// Mitsubishi GX Works2 project: EXC_PLC2   PLC: FX3G

// global labels: Global1
VAR_GLOBAL
  StartBtn AT X001 : BOOL;
  AnalogIn AT D8280 : INT;
  SampledValue AT D2000 : REAL;
  IsRegular AT M50 : BOOL;
  IsPremium AT M51 : BOOL;
  RaspberryStock AT D1100 : REAL;
  LemonStock AT D1110 : REAL;
  StabilizerStock AT D1120 : REAL;
  GummyStock AT D1130 : REAL;
  HasStockRegular AT M80 : BOOL;
  HasStockPremium AT M61 : BOOL;
  HasRaspberryStock AT M222 : BOOL;
  HasLemonStock AT M223 : BOOL;
  HasStabilizerStock AT M224 : BOOL;
  HasGummyStock AT M225 : BOOL;
  HasRasprerryStock1 AT M33 : BOOL;
  HasLemonStock1 AT M34 : BOOL;
  HasStabilizerStock1 AT M35 : BOOL;
  HasGummyStock1 AT M36 : BOOL;
  InvalidOrder AT M66 : BOOL;
  Start_Day AT X007 : BOOL;
  Emergency_Stop AT X005 : BOOL;
  System_On_Lamp AT Y007 : BOOL;
  Analog_Output_Value AT D8282 : INT;
  Produced_Packages_Counter AT D4000 : REAL;  (* מונה מארזים בתחילת כל יום מתאפס לאפס *)
  No_Stock_Error AT M20 : BOOL;
  User_valid AT M12 : BOOL;
  Raspberry_User AT D2100 : REAL;
  Lemon_User AT D2110 : REAL;
  Stabilizer_User AT D2120 : REAL;
  Gummy_User AT D2130 : REAL;
END_VAR
VAR_GLOBAL CONSTANT
  C_R_Raspberry : REAL := 280;
  C_R_Lemon : REAL := 455;
  C_R_Stabilizer : REAL := 105;
  C_P_Raspberry : REAL := 385;
  C_P_Lemon : REAL := 665;
  C_P_Stabilizer : REAL := 210;
  C_R_Gummy : REAL := 28;
  C_P_Gummy : REAL := 70;
END_VAR
VAR_GLOBAL
  PreparationActive AT M101 : BOOL;
  PreparationFinished AT M102 : BOOL;
  CoolingActive AT M103 : BOOL;
  TC50 AT TS50 : BOOL;
  TC80 AT TS80 : BOOL;
  StartMixing AT M2 : BOOL;
  TC2 AT TS2 : BOOL;
  TC1 AT TS1 : BOOL;
END_VAR

// task Task_01 (event TRUE, interval 0, priority 31): POU_01

PROGRAM POU_01
(* structured ladder/FBD written out as ST: instructions are called as NAME(EN, inputs, outputs); _pN, _eN, _tN stand for wires *)
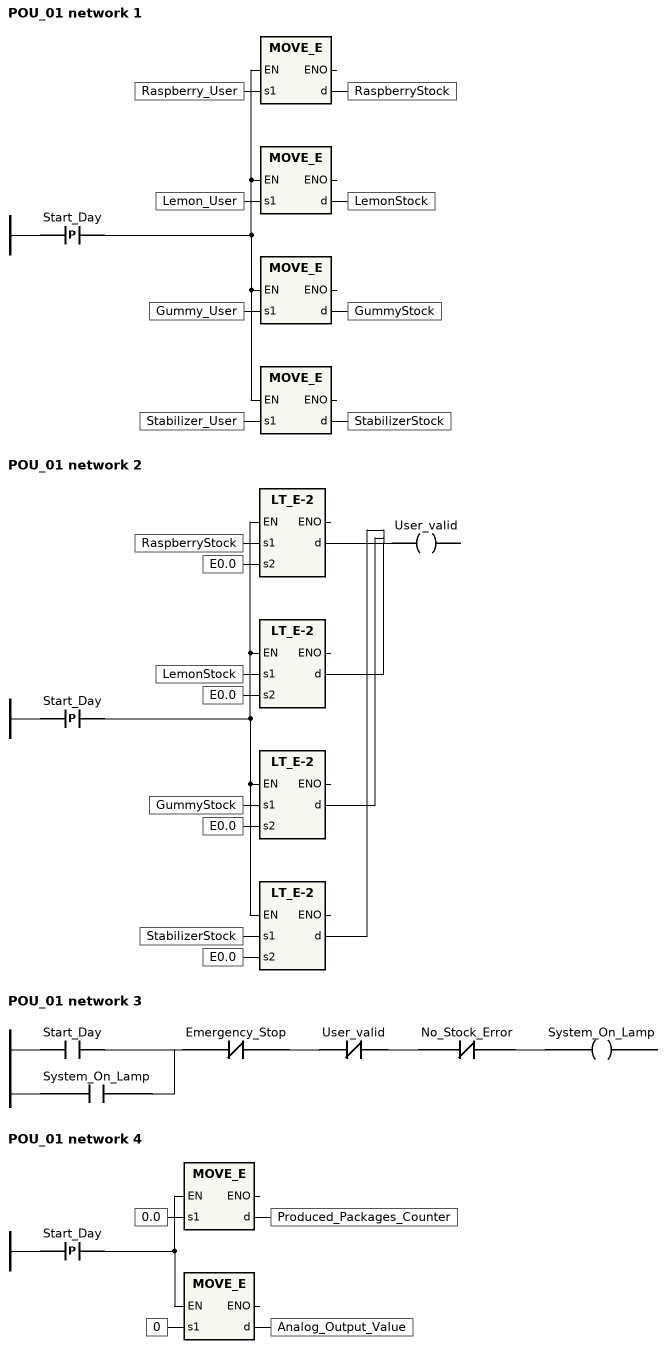
(* network 1 *)
_p1 := LDP(TRUE, Start_Day);
MOVE_E(_p1, Raspberry_User, RaspberryStock);
MOVE_E(_p1, Lemon_User, LemonStock);
MOVE_E(_p1, Gummy_User, GummyStock);
MOVE_E(_p1, Stabilizer_User, StabilizerStock);
(* network 2 *)
_p1 := LDP(TRUE, Start_Day);
LT_E(_p1, RaspberryStock, E0.0, _t2);
LT_E(_p1, LemonStock, E0.0, _t3);
LT_E(_p1, GummyStock, E0.0, _t4);
LT_E(_p1, StabilizerStock, E0.0, _t5);
User_valid := _t2 OR _t3 OR _t4 OR _t5;
(* network 3 *)
System_On_Lamp := (((Start_Day OR System_On_Lamp) AND NOT Emergency_Stop) AND NOT User_valid) AND NOT No_Stock_Error;
(* network 4 *)
_p1 := LDP(TRUE, Start_Day);
MOVE_E(_p1, 0.0, Produced_Packages_Counter);
MOVE_E(_p1, 0, Analog_Output_Value);
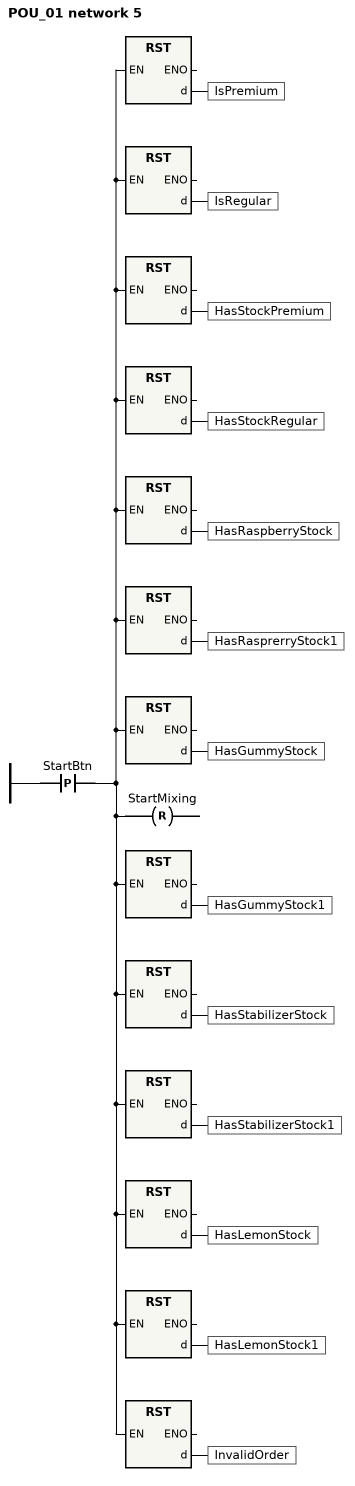
(* network 5 *)
_p1 := LDP(TRUE, StartBtn);
RST(_p1, IsPremium);
RST(_p1, IsRegular);
RST(_p1, HasStockPremium);
RST(_p1, HasStockRegular);
RST(_p1, HasRaspberryStock);
RST(_p1, HasRasprerryStock1);
RST(_p1, HasGummyStock);
RST(_p1, HasGummyStock1);
RST(_p1, HasStabilizerStock);
RST(_p1, HasStabilizerStock1);
RST(_p1, HasLemonStock);
RST(_p1, HasLemonStock1);
RST(_p1, InvalidOrder);
RST(_p1, StartMixing);
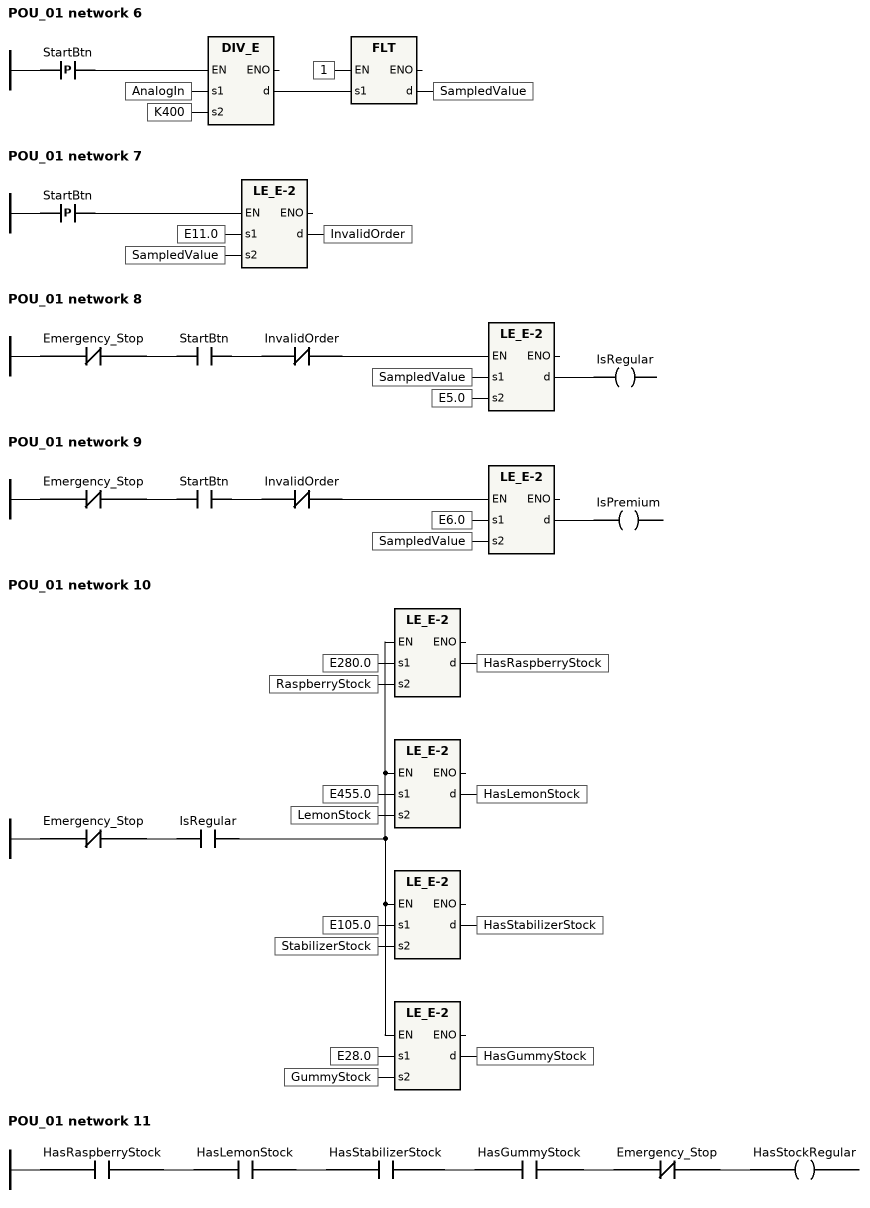
(* network 6 *)
DIV_E(LDP(TRUE, StartBtn), AnalogIn, K400, _t1);
FLT(1, _t1, SampledValue);
(* network 7 *)
LE_E(LDP(TRUE, StartBtn), E11.0, SampledValue, InvalidOrder);
(* network 8 *)
LE_E(NOT Emergency_Stop AND StartBtn AND NOT InvalidOrder, SampledValue, E5.0, _t1);
IsRegular := _t1;
(* network 9 *)
LE_E(NOT Emergency_Stop AND StartBtn AND NOT InvalidOrder, E6.0, SampledValue, _t1);
IsPremium := _t1;
(* network 10 *)
_p1 := NOT Emergency_Stop AND IsRegular;
LE_E(_p1, E280.0, RaspberryStock, HasRaspberryStock);
LE_E(_p1, E455.0, LemonStock, HasLemonStock);
LE_E(_p1, E105.0, StabilizerStock, HasStabilizerStock);
LE_E(_p1, E28.0, GummyStock, HasGummyStock);
(* network 11 *)
HasStockRegular := HasRaspberryStock AND HasLemonStock AND HasStabilizerStock AND HasGummyStock AND NOT Emergency_Stop;
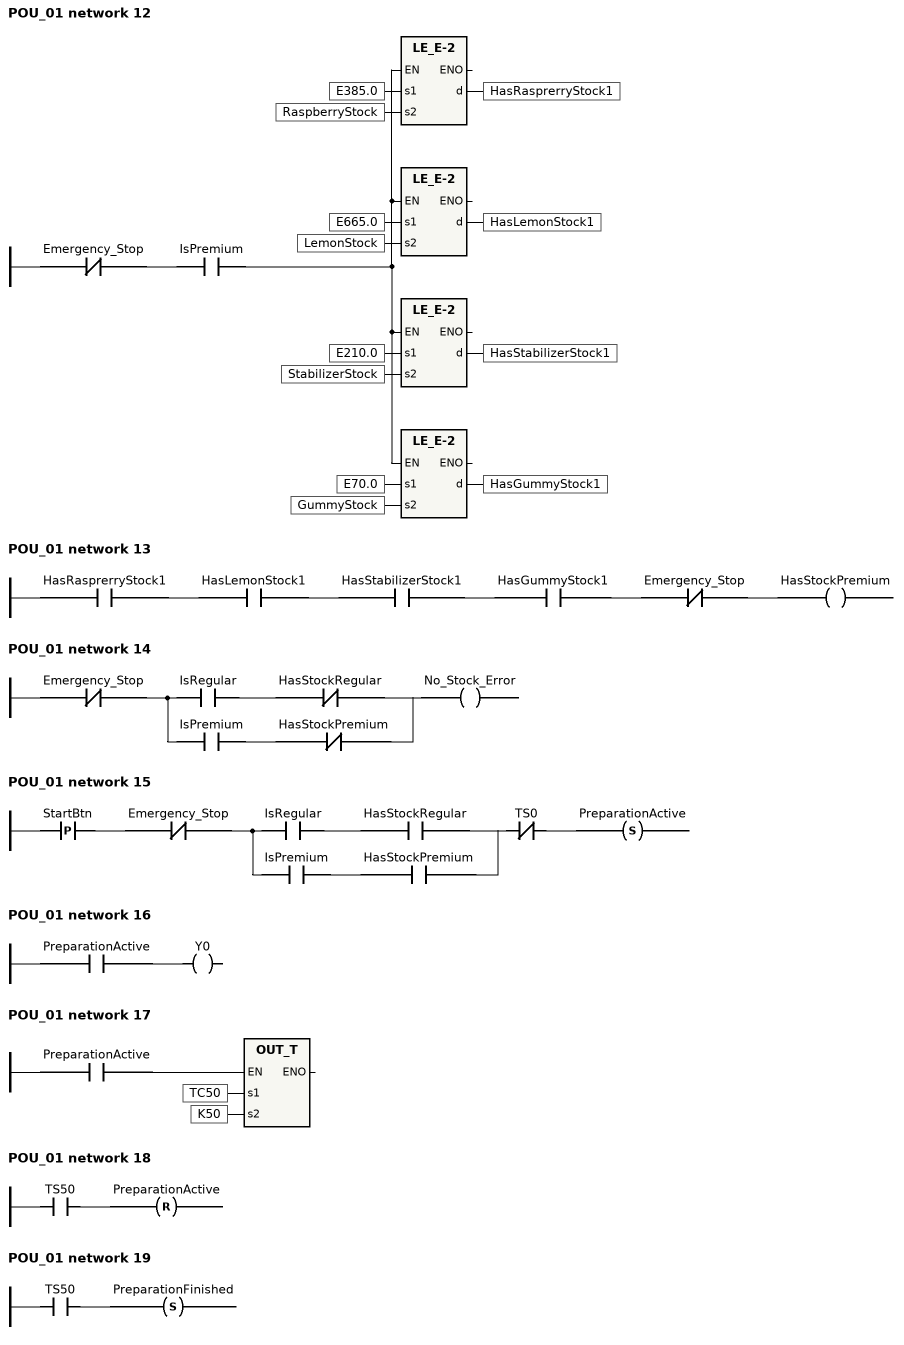
(* network 12 *)
_p1 := NOT Emergency_Stop AND IsPremium;
LE_E(_p1, E385.0, RaspberryStock, HasRasprerryStock1);
LE_E(_p1, E665.0, LemonStock, HasLemonStock1);
LE_E(_p1, E210.0, StabilizerStock, HasStabilizerStock1);
LE_E(_p1, E70.0, GummyStock, HasGummyStock1);
(* network 13 *)
HasStockPremium := HasRasprerryStock1 AND HasLemonStock1 AND HasStabilizerStock1 AND HasGummyStock1 AND NOT Emergency_Stop;
(* network 14 *)
_p1 := NOT Emergency_Stop;
No_Stock_Error := (_p1 AND IsRegular AND NOT HasStockRegular) OR (_p1 AND IsPremium AND NOT HasStockPremium);
(* network 15 *)
_p1 := LDP(TRUE, StartBtn) AND NOT Emergency_Stop;
SET(((_p1 AND IsRegular AND HasStockRegular) OR (_p1 AND IsPremium AND HasStockPremium)) AND NOT TS0, PreparationActive);
(* network 16 *)
Y0 := PreparationActive;
(* network 17 *)
OUT_T(PreparationActive, TC50, K50);
(* network 18 *)
RST(TS50, PreparationActive);
(* network 19 *)
SET(TS50, PreparationFinished);
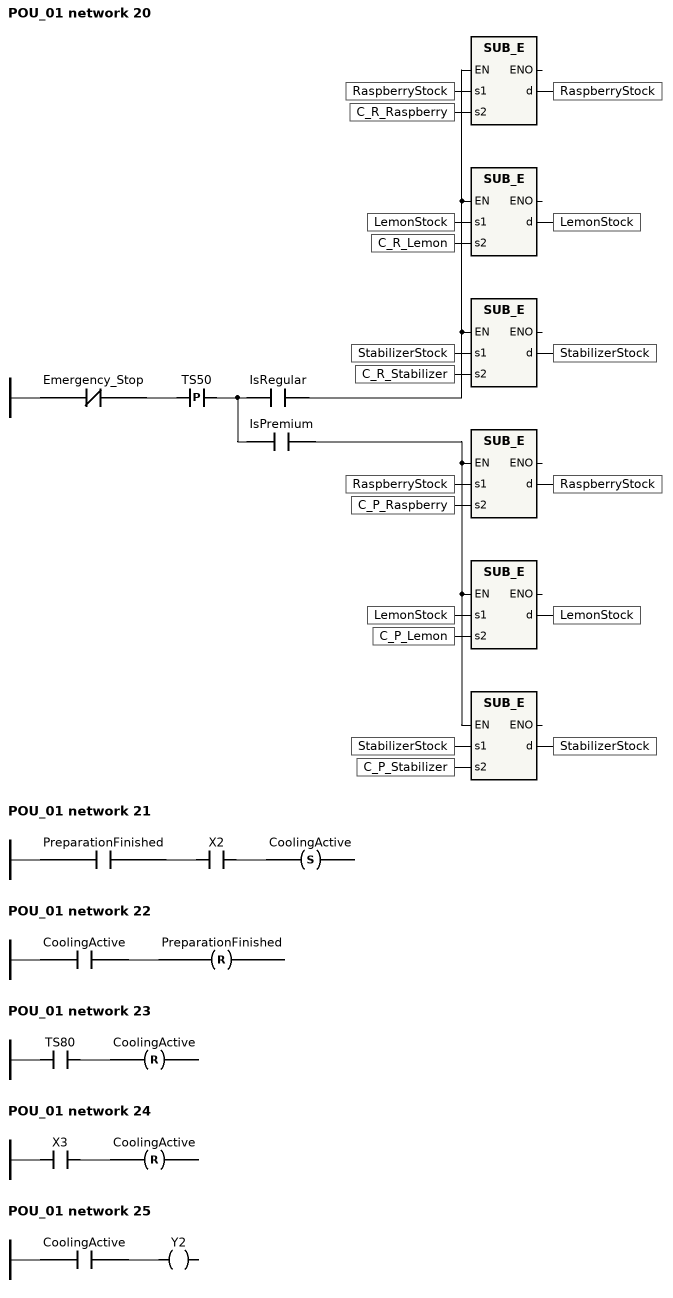
(* network 20 *)
_p1 := NOT Emergency_Stop AND LDP(TRUE, TS50);
_p2 := _p1 AND IsRegular;
SUB_E(_p2, RaspberryStock, C_R_Raspberry, RaspberryStock);
SUB_E(_p2, LemonStock, C_R_Lemon, LemonStock);
SUB_E(_p2, StabilizerStock, C_R_Stabilizer, StabilizerStock);
_p3 := _p1 AND IsPremium;
SUB_E(_p3, RaspberryStock, C_P_Raspberry, RaspberryStock);
SUB_E(_p3, LemonStock, C_P_Lemon, LemonStock);
SUB_E(_p3, StabilizerStock, C_P_Stabilizer, StabilizerStock);
(* network 21 *)
SET(PreparationFinished AND X2, CoolingActive);
(* network 22 *)
RST(CoolingActive, PreparationFinished);
(* network 23 *)
RST(TS80, CoolingActive);
(* network 24 *)
RST(X3, CoolingActive);
(* network 25 *)
Y2 := CoolingActive;
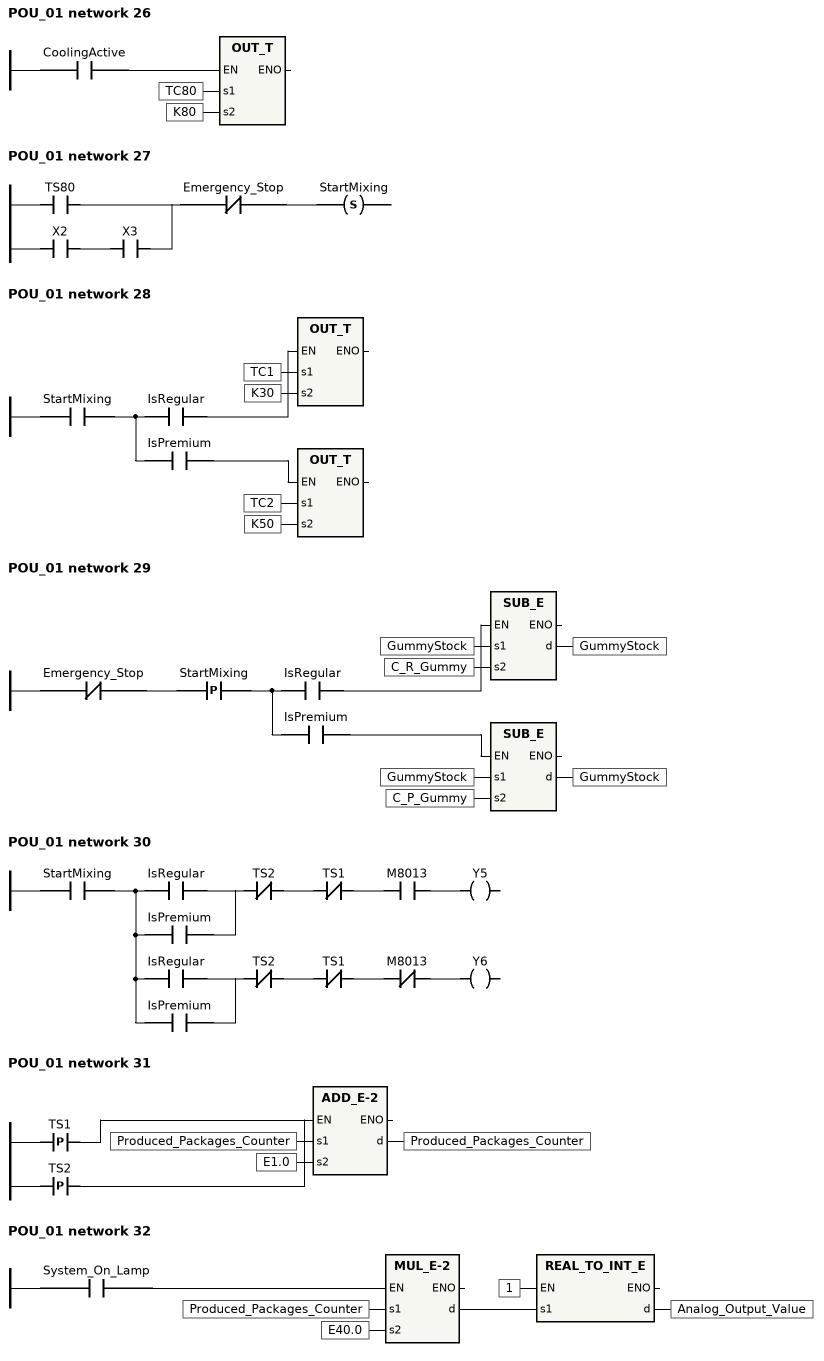
(* network 26 *)
OUT_T(CoolingActive, TC80, K80);
(* network 27 *)
SET((TS80 OR (X2 AND X3)) AND NOT Emergency_Stop, StartMixing);
(* network 28 *)
OUT_T(StartMixing AND IsRegular, TC1, K30);
OUT_T(StartMixing AND IsPremium, TC2, K50);
(* network 29 *)
_p1 := NOT Emergency_Stop AND LDP(TRUE, StartMixing);
SUB_E(_p1 AND IsRegular, GummyStock, C_R_Gummy, GummyStock);
SUB_E(_p1 AND IsPremium, GummyStock, C_P_Gummy, GummyStock);
(* network 30 *)
Y5 := ((((StartMixing AND IsRegular) OR (StartMixing AND IsPremium)) AND NOT TS2) AND NOT TS1) AND M8013;
Y6 := ((((StartMixing AND IsRegular) OR (StartMixing AND IsPremium)) AND NOT TS2) AND NOT TS1) AND NOT M8013;
(* network 31 *)
ADD_E(LDP(TRUE, TS1) OR LDP(TRUE, TS2), Produced_Packages_Counter, E1.0, Produced_Packages_Counter);
(* network 32 *)
MUL_E(System_On_Lamp, Produced_Packages_Counter, E40.0, _t1);
REAL_TO_INT_E(1, _t1, Analog_Output_Value);
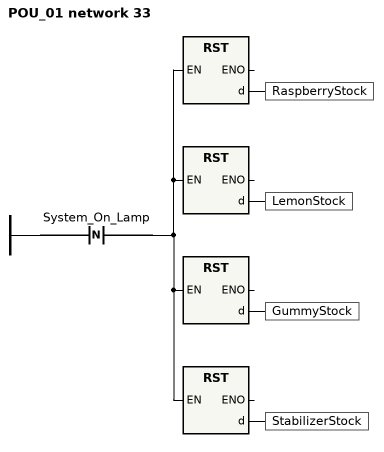
(* network 33 *)
_p1 := LDF(TRUE, System_On_Lamp);
RST(_p1, RaspberryStock);
RST(_p1, LemonStock);
RST(_p1, GummyStock);
RST(_p1, StabilizerStock);
END_PROGRAM
